{attribute 'GeneratedUsingTerminal: CU1521-0010-0000'}
{attribute addProperty BoxType "CU1521-0010-0000"}
{attribute addProperty Id "EtcSlaveTerminalBaseInfoDataAT %I*InfoData_6F19DB2B2"}
{attribute addProperty CRC "2874840167"}
{attribute addProperty Size "2"}
TYPE CU1521_AB5A9467 EXTENDS EtcSlaveTerminalBase :
STRUCT
	{attribute addProperty Name "InfoData"}
	InfoData : InfoData_6F19DB2B;
END_STRUCT
END_TYPE

(* stored: Version 1.2.0.0, ProductVersion 3.1.4024.9
   DUT CU1521_AB5A9467: Id {d1f9224e-402e-47ad-a3d0-f448c59242f6} *)
